PROGRAM INTERNAL PRG_TEST
VAR
END_VAR

END_PROGRAM

(* stored: Version 1.1.0.1, ProductVersion 3.1.4024.11
   POU PRG_TEST: Id {df25c322-66e9-42b5-bf1e-d85a6c4b3bb3}, SpecialFunc None *)
